// TIA Portal project "modbus_tcp_server" (V15)

(* hardware
DEVICE "S7-1200 station_1"  S7-1200 Station
   slot 0: "Rack_0"  S7-1200 Rack  Rack  V1.0
   slot 1: "PLC_1"  CPU 1214C DC/DC/DC  6ES7 214-1AG40-0XB0  V4.2
*)

// ===== PLC "PLC_1"  CPU 1214C DC/DC/DC =====

DATA_BLOCK "tcp_server"   // DB2
{ S7_Optimized_Access := 'TRUE' }
VERSION : 0.1
   VAR
      connect : TCON_IP_v4;
      NDR : Bool;
      DR : Bool;
      ERROR : Bool;
      STATUS : Word;
      DISCONECT : Bool;
   END_VAR
BEGIN
   connect.InterfaceId := 64;
   connect.ID := 1;
   connect.ConnectionType := 11;
   connect.RemoteAddress.ADDR[4] := 123;
   connect.RemoteAddress.ADDR[3] := 0;
   connect.RemoteAddress.ADDR[2] := 168;
   connect.RemoteAddress.ADDR[1] := 192;
   connect.LocalPort := 502;
END_DATA_BLOCK

DATA_BLOCK "data_tcp_server"   // DB3
{ S7_Optimized_Access := 'FALSE' }
VERSION : 0.1
   VAR
      holding_res : Array[0..20] of Int;
   END_VAR
BEGIN
END_DATA_BLOCK

ORGANIZATION_BLOCK "Main"   // OB1, LAD, ProgramCycle
TITLE = "Main Program Sweep (Cycle)"
{ S7_Optimized_Access := 'TRUE' }
VERSION : 0.1
   VAR_INPUT
      Initial_Call : Bool;   // Initial call of this OB
      Remanence : Bool;   // =True, if remanent data are available
   END_VAR
BEGIN

REGION Network 1
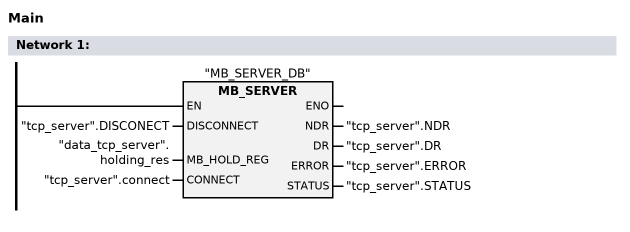
   "MB_SERVER_DB"(DISCONNECT := "tcp_server".DISCONECT,   // MB_SERVER
                  MB_HOLD_REG := "data_tcp_server".holding_res,
                  CONNECT := "tcp_server".connect,
                  NDR => "tcp_server".NDR,
                  DR => "tcp_server".DR,
                  ERROR => "tcp_server".ERROR,
                  STATUS => "tcp_server".STATUS);
END_REGION
END_ORGANIZATION_BLOCK